(* PLC project DataLoggerProject, Industrial Systems DataLogger 2.1, author Developer *)
(* stored: creationDateTime 2024-03-10T08:00:00, organization Industrial Systems, modificationDateTime 2024-03-15T09:45:00, version 2.1 *)

PROGRAM DataLogger
  VAR
    LogCounter : DINT;
    SensorValue : REAL;
    LogEnabled : BOOL;
  END_VAR
  VAR_EXTERNAL
    EXTERNAL_TIMESTAMP : TIME;
  END_VAR

            
IF LogEnabled THEN
    LogCounter := LogCounter + 1;
    (* Attempt to use external logging function *)
    LOG_RECORD(LogCounter, SensorValue);
END_IF;
            
          
END_PROGRAM

CONFIGURATION Config0
  RESOURCE Res0 ON PLC
    TASK Task0(INTERVAL := T#100ms, PRIORITY := 0);
    PROGRAM DataLogger0 WITH Task0 : DataLogger;
  END_RESOURCE
END_CONFIGURATION
